(* PLC project RCP, Beckhoff Automation GmbH TwinCAT PLC Control 3.5.13.21 *)
(* stored: creationDateTime 2024-12-18T13:01:10.755429, modificationDateTime 2024-12-18T13:01:10.759429 *)

(*
:Description: FUNCTION block to control EtherCAT slave device state machine

:Instructions for use: Requires Tc2_EtherCAT Library

Version history:

+-------------+------------+----------------+----------+------------------------------------------+
|Date         | Version    | created under  | Author   | Remark                                   |
+=============+============+================+==========+==========================================+
|2024-12-12   | 1.0.0.0    | 			    | G.P      | Draft					                  |
+-------------+------------+----------------+----------+------------------------------------------+
|			  | 		   | 			    | 		   | Release							      |
+-------------+------------+----------------+----------+------------------------------------------+

*)
FUNCTION_BLOCK FB_SetSlaveState
VAR_INPUT
	sAMSNet		  AT %I*			: AMSNETID; // Linked to EtherCAT master
    nSlaveAddr    AT %I*     		: UINT;	    //  Linked to PortID of slave device
END_VAR
VAR_OUTPUT
END_VAR
VAR
	fbSetECSlaveState				: Tc2_EtherCAT.FB_EcSetSlaveState;
	fbGetECSlaveState				: Tc2_EtherCAT.FB_EcGetSlaveState;
	nState							: UINT;
    sNetId       					: T_AmsNetId; // Must have a value
	_CurrentState					: ST_EcSlaveState;
END_VAR

            
          

METHOD GetState : BOOL
VAR_INPUT
	tTimeout   						: TIME := T#10S; // Timeout time for ECSetSlaveState FB
END_VAR
                  GetState := FALSE;
CASE nState OF
0:
   sNetID := F_CreateAmsNetId( sAMSNet ); // Convert linked EtherCAT Master AMS address and convert to string format FB's can use.
   nState := 1;

1:
  
	// Get slave current state so we can check it changed to the requested state
	fbGetECSlaveState(
		sNetId:= sNetId , 
		nSlaveAddr:= nSlaveAddr, 
		bExecute:= TRUE, 
		tTimeout:= tTimeout);
		nState := 2; // Goto next state
  
2:  
	fbGetECSlaveState(bExecute := FALSE, state=> _CurrentState ); // Reset the execute flag of get slave state
	// Check get slave state has completed without errors
	IF (NOT fbGetECSlaveState.bBusy) AND (NOT fbGetECSlaveState.bError) THEN
		nState := 3; // Move on
	END_IF
3:
   // All complete so reset flags
   GetState := TRUE;
   nState := 0;

100:
   ;                     // Error handling..
END_CASE
                
END_METHOD

METHOD SetState : BOOL
VAR_INPUT
	reqState   						: WORD; // Holds the state the device will be set to 1 = Init, 2 = PreOP, 3 =  Bootstrap, 4 = SafeOp, 8 = OP
    tTimeout   						: TIME := T#10S; // Timeout time for ECSetSlaveState FB
END_VAR
                  SetState := FALSE;
CASE nState OF
0:
   sNetID := F_CreateAmsNetId( sAMSNet ); // Convert linked EtherCAT Master AMS address and convert to string format FB's can use.
   nState := 1;

1:
   // Set the slave to the state requested to goto	
   fbSetECSlaveState(
	sNetId:= sNetId, 
	nSlaveAddr:= nSlaveAddr, // Linked port  
	bExecute:= TRUE , 
	tTimeout:= tTimeout , 
	reqState:= reqState); // State requested to goto
    nState := nState + 1; // Goto next state
2:
  
  fbSetECSlaveState( bExecute := FALSE); // Reset the execute flag of set slave state
  // Check the set slave state has completed without errors
  IF (NOT fbSetECSlaveState.bBusy) AND (NOT fbSetECSlaveState.bError) THEN
	 // Get slave current state so we can check it changed to the requested state
	 fbGetECSlaveState(
		sNetId:= sNetId , 
		nSlaveAddr:= nSlaveAddr, 
		bExecute:= TRUE, 
		tTimeout:= tTimeout);
		nState := 3; // Goto next state
  END_IF
  
  IF fbSetECSlaveState.bError THEN
	  nState := 100;
  END_IF
  
3:  
	fbGetECSlaveState(bExecute := FALSE, state=> _CurrentState ); // Reset the execute flag of get slave state
	// Check get slave state has completed without errors
	IF (NOT fbGetECSlaveState.bBusy) AND (NOT fbGetECSlaveState.bError) THEN
		nState := 4; // Move on
	END_IF
4:
	// Compare requested state with actual state
	CASE (reqState) OF
		  1:
		  	IF _CurrentState.deviceState = Tc2_EtherCAT.EC_DEVICE_STATE_INIT THEN
		  	    nState := 5; // Move to completed state
			END_IF;
		  2:
		  	IF _CurrentState.deviceState = Tc2_EtherCAT.EC_DEVICE_STATE_PREOP THEN
		  	    nState := 5; // Move to completed state
			END_IF;
          4:
		  	IF _CurrentState.deviceState = Tc2_EtherCAT.EC_DEVICE_STATE_SAFEOP THEN
		  	    nState := 5; // Move to completed state
			END_IF;
		  8:
		  	IF _CurrentState.deviceState = Tc2_EtherCAT.EC_DEVICE_STATE_OP THEN
		  	    nState := 5; // Move to completed state
			END_IF;
	  END_CASE
5:
   // All complete so reset flags
   SetState := TRUE;
   nState := 0;

100:
   ;                     // Error handling..
END_CASE
                
END_METHOD

METHOD ResetStateToOp : BOOL
VAR_INPUT
    tTimeout   						: TIME := T#10S; // Timeout time for ECSetSlaveState FB
END_VAR
                  ResetStateToOp := FALSE;
CASE nState OF
0:
   sNetID := F_CreateAmsNetId( sAMSNet ); // Convert linked EtherCAT Master AMS address and convert to string format FB's can use.
   nState := 1;

1:
   // Set the slave to the state requested to goto	
   fbSetECSlaveState(
	sNetId:= sNetId, 
	nSlaveAddr:= nSlaveAddr, // Linked port  
	bExecute:= TRUE , 
	tTimeout:= tTimeout , 
	reqState:= 1); // State requested to init
    nState := nState + 1; // Goto next state
2:
  
  fbSetECSlaveState( bExecute := FALSE); // Reset the execute flag of set slave state
  // Check the set slave state has completed without errors
  IF (NOT fbSetECSlaveState.bBusy) AND (NOT fbSetECSlaveState.bError) THEN
	 // Get slave current state so we can check it changed to the requested state
	 fbGetECSlaveState(
		sNetId:= sNetId , 
		nSlaveAddr:= nSlaveAddr, 
		bExecute:= TRUE, 
		tTimeout:= tTimeout);
		nState := 3; // Goto next state
  END_IF
  
  IF fbSetECSlaveState.bError THEN
	  nState := 100;
  END_IF
  
3:  
	fbGetECSlaveState(bExecute := FALSE, state=> _CurrentState ); // Reset the execute flag of get slave state
	// Check get slave state has completed without errors
	IF (NOT fbGetECSlaveState.bBusy) AND (NOT fbGetECSlaveState.bError) THEN
		nState := 4; // Move on
	END_IF
	
4:
	// Make sure in correct state
  	IF _CurrentState.deviceState = Tc2_EtherCAT.EC_DEVICE_STATE_INIT THEN
  	    nState := 5; // Move to completed state
	END_IF;
	
5:
	// Set the slave to the state requested to goto	
   fbSetECSlaveState(
	sNetId:= sNetId, 
	nSlaveAddr:= nSlaveAddr, // Linked port  
	bExecute:= TRUE , 
	tTimeout:= tTimeout , 
	reqState:= 8); // State requested to OP
    nState := nState + 1; // Goto next state
	
6:
	fbSetECSlaveState( bExecute := FALSE); // Reset the execute flag of set slave state
  	// Check the set slave state has completed without errors
  	IF (NOT fbSetECSlaveState.bBusy) AND (NOT fbSetECSlaveState.bError) THEN
		// Get slave current state so we can check it changed to the requested state
	 	fbGetECSlaveState(
			sNetId:= sNetId , 
			nSlaveAddr:= nSlaveAddr, 
			bExecute:= TRUE, 
			tTimeout:= tTimeout);
			nState := 7; // Goto next state
  	END_IF
  
	IF fbSetECSlaveState.bError THEN
		nState := 100;
  	END_IF
	
7:  
  	fbGetECSlaveState(bExecute := FALSE, state=> _CurrentState ); // Reset the execute flag of get slave state
	// Check get slave state has completed without errors
	IF (NOT fbGetECSlaveState.bBusy) AND (NOT fbGetECSlaveState.bError) THEN
		nState := 8; // Move on
	END_IF
	
8:
	// Compare requested state with actual state
  	IF _CurrentState.deviceState = Tc2_EtherCAT.EC_DEVICE_STATE_OP THEN
  	    nState := 9; // Move to completed state
	END_IF;
	
9:
   // All complete so reset flags
   ResetStateToOp := TRUE;
   nState := 0;

100:
   ;                     // Error handling..
END_CASE
                
END_METHOD

PROPERTY CurrentState : ST_EcSlaveState
GET
VAR
END_VAR
                    CurrentState := _CurrentState;
                  
END_GET
END_PROPERTY
END_FUNCTION_BLOCK
